FUNCTION_BLOCK E_D_FF (* Event-driven Data(D)Latch *)
  (* Standard: 61499-1; Classification: Event processing *)
  (* Version 0.2, 2003-12-30, JHC, Rockwell Automation, Updated for 61499-1 CDV. *)
  (* Version 0.1, 2002-01-29, JHC, Rockwell Automation, XML version *)
  (* Version 0.0, 2000-03-12, JHC, Rockwell Automation, SRC version *)
  (* Compiler header: package fb.rt.events; *)
  (* Compiler Java IBM VisualAge 3.0 *)
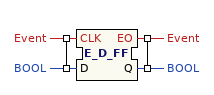
  EVENT_INPUT
    CLK WITH D; (* Data Clock *)
  END_EVENT
  EVENT_OUTPUT
    EO WITH Q; (* Output Event when Q output changes *)
  END_EVENT
  VAR_INPUT
    D : BOOL; (* Data Input *)
  END_VAR
  VAR_OUTPUT
    Q : BOOL; (* Latched Data *)
  END_VAR
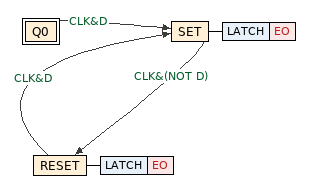
  EC_STATES
    Q0; (* Q is FALSE initially *)
    RESET : LATCH -> EO; (* Reset Q and issue EO *)
    SET : LATCH -> EO; (* Latch and issue EO *)
  END_STATES
  EC_TRANSITIONS
    Q0 TO SET := CLK&D;
    SET TO RESET := CLK&(NOT D);
    RESET TO SET := CLK&D;
  END_TRANSITIONS
  ALGORITHM LATCH IN ST:
Q:=D;
  END_ALGORITHM
END_FUNCTION_BLOCK
